Fanuc KAREL source: ko00038.KL

-- PROVISIONAL review KL for V770-1; original PC SHA256 ebf2edf1f8195e34f504514f1ee030d5fc6f057452e726ab470a0e72e263f8f7
-- Incomplete behavior may be omitted. Consult companion uncertainty JSON. Do not deploy.
PROGRAM KO00038
%NOLOCKGROUP
BEGIN
  -- UNRESOLVED_PC offsets 5-12; opcodes 9D,23
  -- UNRESOLVED_PC offsets 17-69; opcodes 27,27,49,7E,AD,27,49,7E,AD,22,31,7E,4A
  -- UNRESOLVED_PC offsets 74-78; opcodes 7F
END KO00038
